{attribute 'qualified_only'}
VAR_GLOBAL
    //Timers
    tDriveHomeToStation : TON := (PT := T#15S);   //car ride
    tWalkHomeToStation : TON := (PT := T#10S);    //walking
    tWalkStationToSchool : TON := (PT := T#8S);   // walking
	Timer : TON;								  //trainride

    //starting signals
    bStartDrive : BOOL := FALSE;
    bStartWalk1 : BOOL := FALSE;
    bStartTrain : BOOL := FALSE;
    bStartWalk2 : BOOL := FALSE;
    InternalStart : BOOL;
	
    //State machine
    Step : INT := 0;

    //Info-output
    sStatus : STRING;
END_VAR

(* stored: Version 1.1.0.1, ProductVersion 3.1.4024.15
   GVL GVL: Id {82520393-6125-4684-a7fb-71ff98d41678} *)
